FUNCTION WithinTolerance : BOOL
VAR_INPUT
	v1 : LREAL;
	v2 : LREAL;
	tolerance : LREAL;
END_VAR

WithinTolerance := ABS(v1-v2) < tolerance;

END_FUNCTION

(* stored: Version 1.1.0.1, ProductVersion 3.1.4024.11
   POU WithinTolerance: Id {b9c242fe-198a-4c23-ab60-1ac81842e68f}, SpecialFunc None *)
